// TIA Portal V17 export
VAR_GLOBAL   // PLC tag table "Convoyeur"
   Start_Button AT %I0.0 : Bool;   // Bouton marche
   Stop_Button AT %I0.1 : Bool;
   Lamp AT %Q0.0 : Bool;
   Speed_Display AT %MD20 : Real;   //    {ExternalWritable false}
END_VAR
VAR_GLOBAL CONSTANT   // user constants
   MaxStarts : Int := 1000;
END_VAR
